{attribute 'qualified_only'}
{attribute 'strict'}
TYPE E_MbAddressing :
(
	Modicon := 0,
	Offset0,
	Offset1
);
END_TYPE

(* stored: Version 1.1.0.1
   DUT E_MbAddressing: Id {1508dbc4-6629-40b8-8cab-7ef8fa791287} *)
